PROGRAM PRG_TaktGen
VAR
	fb_TaktGen	: FB_Takt;
END_VAR

fb_TaktGen();

END_PROGRAM

(* stored: Version 1.1.0.1, ProductVersion 3.1.4024.12
   POU PRG_TaktGen: Id {2c3c58b0-390f-4f6a-8943-f24fb69e5626}, SpecialFunc None *)
